SUBAPPLICATION Softkey_IE_1 (* 1 SoftKey-Objekt, liest ein konfigurierbares Event (SoftKeyActivationCode, z.B. SK_PRESSED/SK_RELEASED) als reines IND-Event - duenner Wrapper um Softkey_IE (Konvention in diesem Projekt: Softkey_IE wird nie roh inline verwendet, immer gewrappt). *)
  (* Standard: 61499-2 *)
  (* Version 1.0, 2026-09-11, Franz Höpfinger, initial implementation *)
  PACKAGE MyLib::sys;
  IMPORT isobus::UT::Q::const::IDs::ID_NULL;
  IMPORT isobus::UT::io::Softkey::SoftKeyActivationCode::Invalid;
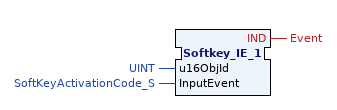
  EVENT_OUTPUT
    IND; (* Feuert wenn das konfigurierte InputEvent auftritt *)
  END_EVENT
  VAR_INPUT
    u16ObjId : UINT := ID_NULL; (* Object ID SoftKey *)
    InputEvent : isobus::UT::io::Softkey::SoftKeyActivationCode_S := Invalid; (* z.B. SK_PRESSED, SK_RELEASED *)
  END_VAR
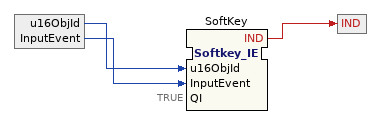
  FBS
    SoftKey : isobus::UT::io::Softkey::Softkey_IE(QI := TRUE);
  END_FBS
  EVENT_CONNECTIONS
    SoftKey.IND TO IND;
  END_CONNECTIONS
  DATA_CONNECTIONS
    u16ObjId TO SoftKey.u16ObjId;
    InputEvent TO SoftKey.InputEvent;
  END_CONNECTIONS
END_SUBAPPLICATION
